FUNCTION_BLOCK CSV_WRITER_10
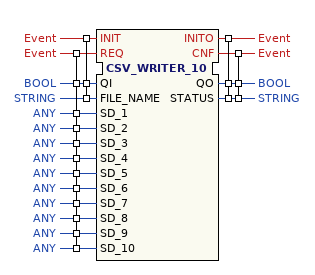
  EVENT_INPUT
    INIT WITH QI, FILE_NAME;
    REQ WITH QI, SD_1, SD_2, SD_3, SD_4, SD_5, SD_6, SD_7, SD_8, SD_9, SD_10;
  END_EVENT
  EVENT_OUTPUT
    INITO WITH QO, STATUS;
    CNF WITH QO, STATUS;
  END_EVENT
  VAR_INPUT
    QI : BOOL;
    FILE_NAME : STRING;
    SD_1 : ANY;
    SD_2 : ANY;
    SD_3 : ANY;
    SD_4 : ANY;
    SD_5 : ANY;
    SD_6 : ANY;
    SD_7 : ANY;
    SD_8 : ANY;
    SD_9 : ANY;
    SD_10 : ANY;
  END_VAR
  VAR_OUTPUT
    QO : BOOL;
    STATUS : STRING;
  END_VAR
END_FUNCTION_BLOCK
